# EPICS autosave request: iocBoot/sioc-esb-xps5/xps.req
file xpsm.req P=ESB:XPS5:m1
file xpsm.req P=ESB:XPS5:m2
file xpsm.req P=ESB:XPS5:m3
file xpsm.req P=ESB:XPS5:m4
file xpsm.req P=ESB:XPS5:m5
file xpsm.req P=ESB:XPS5:m6
file xpsm.req P=ESB:XPS5:m7
file xpsm.req P=ESB:XPS5:m8
